(*
SPDX-FileCopyrightText: © 2026 Oleksandr Tiutyk <trofimich@gmail.com>
SPDX-License-Identifier: MIT
License: https://opensource.org/license/mit
*)

(*!
<summary>
Internal service program providing access to the current library namespace.
</summary>
*)

{attribute 'no_explicit_call' := 'do not call this POU directly'}
PROGRAM INTERNAL CurrentNamespace
VAR
	{attribute 'hide'} 
	_NamespaceExtractor : NamespaceExtractor;
END_VAR

(*!
<summary>Borrows the compiler-initialized namespace buffer for the program lifetime.</summary>
<description>
Callers must not modify or retain the reference beyond the program lifetime. A reference property remains
technically writable without a setter; read-only use is a caller obligation. No allocation or initialization occurs.
</description>
*)
{attribute 'monitoring' := 'call'}
PROPERTY Name : REFERENCE TO STRING
GET
Name REF= _NamespaceExtractor.CurrentNamespace;
END_GET
END_PROPERTY

END_PROGRAM

(* stored: Version 1.1.0.1, ProductVersion 3.1.4026.20
   POU CurrentNamespace: Id {506615aa-524b-4ab8-910f-0aebdcb95c3f}, SpecialFunc None
   Property Name: Id {48dc4841-9c00-4a7f-a2e0-77db98a8158a}
   Get Get: Id {832d31e5-67f0-4f0f-a948-2ec7f998fc90} *)
